FUNCTION_BLOCK FINAL FB_TwinSAFE EXTENDS FB_EventLogger
VAR_IN_OUT
	Control								: ST_System;
END_VAR
VAR
	_ComErr					AT %I*		: BOOL;
	_FbErr					AT %I*		: BOOL;
	_OutErr					AT %I*		: BOOL;
	_ComStartUp				AT %I*		: BOOL;
	_OtherErr				AT %I*		: BOOL;
	_State					AT %I*		: UINT;
	_Daig					AT %I*		: UINT;
	_FSOUTModule1Fault 		AT %I* 		: BOOL;
	_FSOUTModule2Fault 		AT %I* 		: BOOL;
	_FSOUTModule3Fault 		AT %I* 		: BOOL;
	_FSOUTModule4Fault 		AT %I* 		: BOOL;
	_FSOUTModule5Fault 		AT %I* 		: BOOL;
	_FSOUTModule6Fault 		AT %I* 		: BOOL;
	_FSOUTRelaisModuleFault AT %I*      : BOOL;
	_FSINModule1Fault		AT %I* 		: BOOL;
	_FSINModule2Fault		AT %I* 		: BOOL;
	_FSINModule3Fault		AT %I* 		: BOOL;
	_FSINModule4Fault		AT %I* 		: BOOL;
	_FSINModule5Fault		AT %I* 		: BOOL;
	_FSINModule6Fault		AT %I* 		: BOOL;
	_FSINModule7Fault		AT %I* 		: BOOL;
	_FSINModule8Fault		AT %I* 		: BOOL;
	_FSINModule9Fault		AT %I* 		: BOOL;
	_FSINModule10Fault		AT %I* 		: BOOL;
	_SafetyChainFault 	    AT %I*  	: BOOL;
	_SafetyInRun			AT %I*  	: BOOL;
	_Module1Fault			AT %I*  	: BOOL;
	_RunStop				AT %Q*		: BOOL;
	_ErrAck					AT %Q*		: BOOL;
	_SafetyInRunReturn		AT %Q*  	: BOOL;
	_ModuleFault					  	: BOOL;
	_Alarm								: BOOL;					
	_Warning							: BOOL;					
	_AlarmMute							: BOOL;					
	_AlarmNum							: DINT;					
	_WarningNum							: DINT;					
	_FaultTimer_ET						: REAL;	
	_r_Trig								: ARRAY[0..9] OF R_TRIG;
END_VAR
VAR PERSISTENT
	_Name								: STRING[15];				//Name for HMI
	_Description						: STRING[40];				//Description for HMI
	_FaultTimer_PT						: REAL;						//Fault timer preset time
END_VAR

M_Control();
M_AlarmMonitor();
M_WarningMonitor();

//Alarm mute reset
IF Control.Inputs.AlarmMuteReset THEN _AlarmMute := FALSE; END_IF

{attribute 'monitoring' := 'variable'}
PROPERTY PUBLIC Alarm : Bool
GET
Alarm := _Alarm;
END_GET
END_PROPERTY

{attribute 'monitoring' := 'variable'}
PROPERTY PUBLIC Description : String[40]
GET
Description := _Description;
END_GET
SET
_Description := Description;
END_SET
END_PROPERTY

{attribute 'monitoring' := 'variable'}
PROPERTY PUBLIC FaultTimer_ET : real
GET
FaultTimer_ET := _FaultTimer_ET;
END_GET
END_PROPERTY

{attribute 'monitoring' := 'variable'}
PROPERTY PUBLIC FaultTimer_PT : real
GET
FaultTimer_PT := _FaultTimer_PT;
END_GET
SET
_FaultTimer_PT := FaultTimer_PT;
END_SET
END_PROPERTY

METHOD PRIVATE M_AlarmMonitor
VAR_INPUT
END_VAR
VAR_INST
END_VAR
VAR_INST // added by the converter: edge detectors and wires of the graphical bodies
    _w1, _w2, _w3 : BOOL;
END_VAR
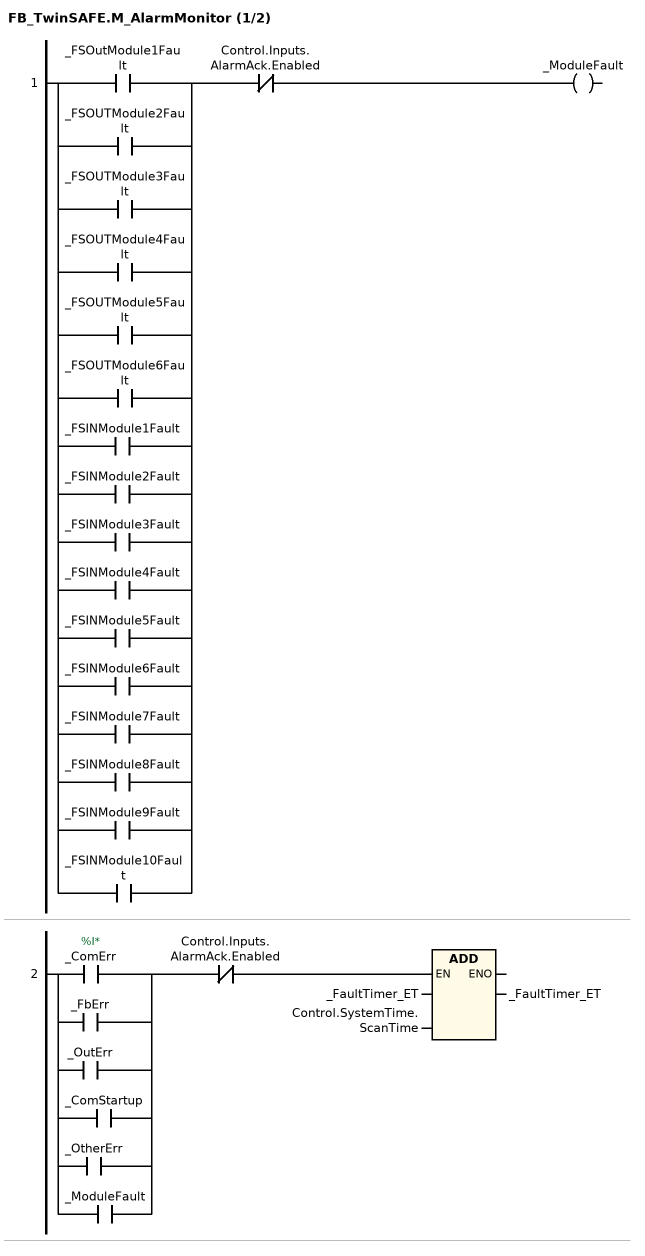
// NETWORK 1
_ModuleFault := (_FSOutModule1Fault OR _FSOUTModule2Fault OR _FSOUTModule3Fault OR _FSOUTModule4Fault OR _FSOUTModule5Fault OR _FSOUTModule6Fault OR _FSINModule1Fault OR _FSINModule2Fault OR _FSINModule3Fault OR _FSINModule4Fault OR _FSINModule5Fault OR _FSINModule6Fault OR _FSINModule7Fault OR _FSINModule8Fault OR _FSINModule9Fault OR _FSINModule10Fault) AND NOT Control.Inputs.AlarmAck.Enabled;

// NETWORK 2
//   _ComErr: AT %I*
//   _FaultTimer_ET: Fault timer elapsed
//   Control.SystemTime.ScanTime: Last scan time (Seconds)
IF (_ComErr OR _FbErr OR _OutErr OR _ComStartup OR _OtherErr OR _ModuleFault) AND NOT Control.Inputs.AlarmAck.Enabled THEN
    _FaultTimer_ET := _FaultTimer_ET + Control.SystemTime.ScanTime;
END_IF

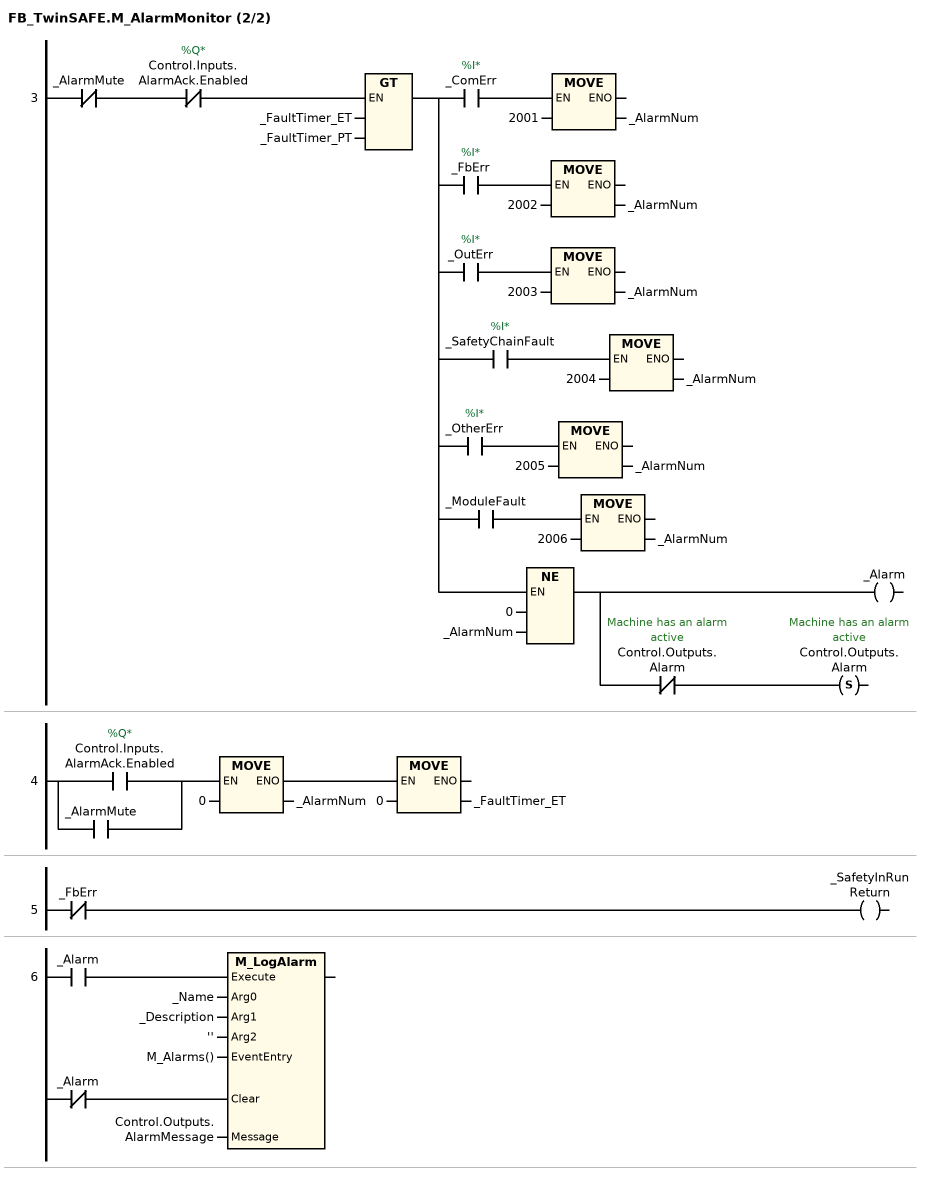
// NETWORK 3
//   Control.Inputs.AlarmAck.Enabled: AT %Q*
//   _ComErr: AT %I*
//   _FbErr: AT %I*
//   _OutErr: AT %I*
//   _SafetyChainFault: AT %I*
//   _OtherErr: AT %I*
//   Control.Outputs.Alarm: Machine has an alarm active
_w1 := NOT _AlarmMute AND NOT Control.Inputs.AlarmAck.Enabled AND _FaultTimer_ET > _FaultTimer_PT;
IF _w1 AND _ComErr THEN _AlarmNum := 2001; END_IF
IF _w1 AND _FbErr THEN _AlarmNum := 2002; END_IF
IF _w1 AND _OutErr THEN _AlarmNum := 2003; END_IF
IF _w1 AND _SafetyChainFault THEN _AlarmNum := 2004; END_IF
IF _w1 AND _OtherErr THEN _AlarmNum := 2005; END_IF
IF _w1 AND _ModuleFault THEN _AlarmNum := 2006; END_IF
_w2 := _w1 AND 0 <> _AlarmNum;
_Alarm := _w2;
Control.Outputs.Alarm S= _w2 AND NOT Control.Outputs.Alarm;

// NETWORK 4
//   Control.Inputs.AlarmAck.Enabled: AT %Q*
_w3 := Control.Inputs.AlarmAck.Enabled OR _AlarmMute;
IF _w3 THEN _AlarmNum := 0; END_IF
IF _w3 THEN _FaultTimer_ET := 0; END_IF

// NETWORK 5
_SafetyInRunReturn := NOT _FbErr;

// NETWORK 6
M_LogAlarm(Execute := _Alarm, Arg0 := _Name, Arg1 := _Description, Arg2 := '', EventEntry := M_Alarms(), Clear := NOT _Alarm, Message := Control.Outputs.AlarmMessage);
END_METHOD

METHOD PRIVATE M_Alarms : TcEventEntry
VAR_INPUT
END_VAR
VAR_INST
END_VAR
CASE _AlarmNum OF		
2001:	M_Alarms := 	TC_Events.TcTwinSafe.A_2001;//Communication Error			
2002:	M_Alarms := 	TC_Events.TcTwinSafe.A_2002;//Feedback Error			
2003:	M_Alarms := 	TC_Events.TcTwinSafe.A_2003;//Output Error	
2004:	M_Alarms := 	TC_Events.TcTwinSafe.A_2004;//Safety Chain Fault	    
2005:	M_Alarms := 	TC_Events.TcTwinSafe.A_2005;//Other Error	 
2006:	M_Alarms := 	TC_Events.TcTwinSafe.A_2006;//Module Error	                    	
ELSE                        	
		M_Alarms := 	TC_Events.TcTwinSafe.A_Undefined;
END_CASE
END_METHOD

METHOD PRIVATE M_Control
VAR_INPUT
END_VAR
VAR_INST
	_resetStep				: INT;
END_VAR
VAR_INST // added by the converter: edge detectors and wires of the graphical bodies
    _rt1 : R_TRIG;
    _w1 : BOOL;
END_VAR
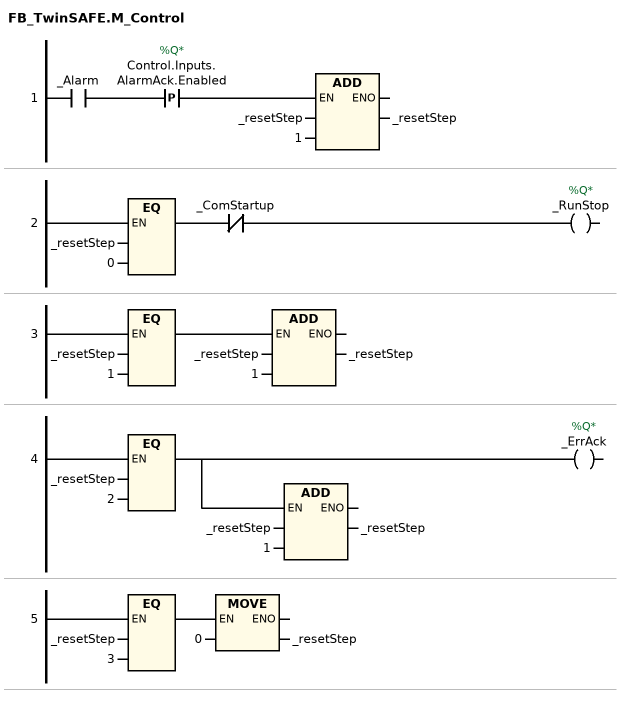
// NETWORK 1
//   Control.Inputs.AlarmAck.Enabled: AT %Q*
_rt1(CLK := Control.Inputs.AlarmAck.Enabled);
IF _Alarm AND _rt1.Q THEN _resetStep := _resetStep + 1; END_IF

// NETWORK 2
//   _RunStop: AT %Q*
_RunStop := _resetStep = 0 AND NOT _ComStartup;

// NETWORK 3
IF _resetStep = 1 THEN _resetStep := _resetStep + 1; END_IF

// NETWORK 4
//   _ErrAck: AT %Q*
_w1 := _resetStep = 2;
_ErrAck := _w1;
IF _w1 THEN _resetStep := _resetStep + 1; END_IF

// NETWORK 5
IF _resetStep = 3 THEN _resetStep := 0; END_IF
END_METHOD

METHOD PRIVATE M_WarningMonitor
VAR_INPUT
END_VAR
VAR_INST
END_VAR
VAR_INST // added by the converter: edge detectors and wires of the graphical bodies
    _w1, _w2 : BOOL;
END_VAR
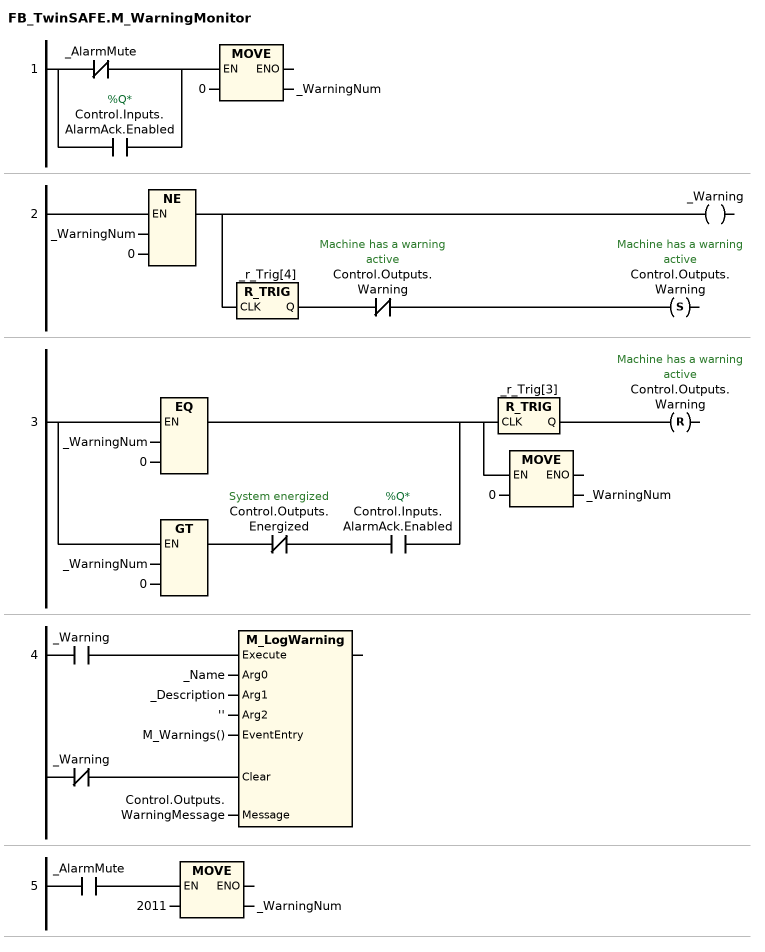
// NETWORK 1
//   Control.Inputs.AlarmAck.Enabled: AT %Q*
IF NOT _AlarmMute OR Control.Inputs.AlarmAck.Enabled THEN _WarningNum := 0; END_IF

// NETWORK 2
//   Control.Outputs.Warning: Machine has a warning active
_w1 := _WarningNum <> 0;
_Warning := _w1;
_r_Trig[4](CLK := _w1); // R_TRIG
Control.Outputs.Warning S= _r_Trig[4].Q AND NOT Control.Outputs.Warning;

// NETWORK 3
//   Control.Outputs.Energized: System energized
//   Control.Inputs.AlarmAck.Enabled: AT %Q*
//   Control.Outputs.Warning: Machine has a warning active
_w2 := _WarningNum = 0 OR _WarningNum > 0 AND NOT Control.Outputs.Energized AND Control.Inputs.AlarmAck.Enabled;
_r_Trig[3](CLK := _w2); // R_TRIG
Control.Outputs.Warning R= _r_Trig[3].Q;
IF _w2 THEN _WarningNum := 0; END_IF

// NETWORK 4
M_LogWarning(Execute := _Warning, Arg0 := _Name, Arg1 := _Description, Arg2 := '', EventEntry := M_Warnings(), Clear := NOT _Warning, Message := Control.Outputs.WarningMessage);

// NETWORK 5
IF _AlarmMute THEN _WarningNum := 2011; END_IF
END_METHOD

METHOD PRIVATE M_Warnings : TcEventEntry
VAR_INPUT
END_VAR
VAR_INST
END_VAR
CASE _WarningNum OF
	2011:   M_Warnings :=	TC_Events.TcTwinSafe.W_2011;//Alarm Mute Active			
ELSE
	M_Warnings := 	TC_Events.TcTwinSafe.W_Undefined;
END_CASE
END_METHOD

{attribute 'monitoring' := 'variable'}
PROPERTY PUBLIC Name : String[15]
GET
Name := _Name;
END_GET
SET
_Name := Name;
END_SET
END_PROPERTY

{attribute 'monitoring' := 'variable'}
PROPERTY PUBLIC Warning : Bool
GET
Warning := _Warning;
END_GET
END_PROPERTY

END_FUNCTION_BLOCK

(* stored: Version 1.1.0.1, ProductVersion 3.1.4024.3
   POU FB_TwinSAFE: Id {47e72a5f-2a61-41d0-8001-1770deb34dd1}, SpecialFunc None
   Property Alarm: Id {d6591078-7152-47be-9847-56e7ed24d89c}
   Get Get: Id {58654c60-ac8e-45ed-8df3-b26800e4491b}
   Property Description: Id {88588e26-3527-42eb-8c91-025c666c8b6a}
   Get Get: Id {0e5d68c3-ee79-406b-b721-149c84040c88}
   Set Set: Id {73182e88-51a5-4599-b023-614c633b4246}
   Property FaultTimer_ET: Id {c8dfdc42-a2e4-4521-b182-bf9a3679b7d6}
   Get Get: Id {23e3c838-fdf2-496b-8fa4-d0ee0c743a02}
   Property FaultTimer_PT: Id {5d80a0f5-1676-4b2a-a136-894530196502}
   Get Get: Id {3c1cf4e5-60a5-40c0-890e-d60cda1948ff}
   Set Set: Id {da3ebae9-e3d0-47fd-8654-566150b6b6bc}
   Method M_AlarmMonitor: Id {4ae8289e-ec8b-473f-b170-ca3ec84cf5ec}
   Method M_Alarms: Id {442ff02a-e34e-415f-86e0-78bb026ecca4}
   Method M_Control: Id {42f3880a-736c-45da-9415-e92bcb10a54c}
   Method M_WarningMonitor: Id {a7412c32-e8f2-4631-8b0e-097a9acd0692}
   Method M_Warnings: Id {bca6d6e2-b4bb-451e-8798-c721eb93a549}
   Property Name: Id {e44063aa-aa11-4d90-928f-e9c14fbace65}
   Get Get: Id {95b72992-f853-48e5-882d-3bcc79eeb03a}
   Set Set: Id {ee23b637-3601-4ac7-9d5d-a566ff0c0be8}
   Property Warning: Id {37ccfa29-ba0e-4236-a681-f49a0a573728}
   Get Get: Id {68260024-7447-4a6a-8ad3-3840e737a4ec} *)
